// TIA Portal V17 export
// export: Created 2026-04-13T11:12:43.5207682Z, ExportSetting WithDefaults, DisplayName Totally Integrated Automation Portal, DisplayVersion V17 Update 4, DisplayName TIA Portal Openness, DisplayVersion V17 Update 4, DisplayName TIA Portal Version Control Interface, DisplayVersion V17, DisplayName SINAMICS Startdrive Advanced, DisplayVersion V17, DisplayName SINAMICS Startdrive G130, G150, S120, S150, SINAMICS MV, S210, DisplayVersion V17, DisplayName SINAMICS Startdrive G110M, G120, G120C, G120D, G120P, G115D, DisplayVersion V17, DisplayName STEP 7 Professional, DisplayVersion V17 Update 4, DisplayName STEP 7 Safety, DisplayVersion V17, DisplayName WinCC Professional, DisplayVersion V17 Update 4
FUNCTION_BLOCK "12放空阀"   // FB8, SCL
{ S7_Optimized_Access := 'FALSE' }
VERSION : 0.1
// stored: AutoNumber true, IsIECCheckEnabled false, SetENOAutomatically false, UDAEnableTagReadback false
   VAR_INPUT
      条件1 : Real;
      工程上限 : Real;
      工程下限 : Real;
      模拟高限 : Int;
      模拟低限 : Int;
   END_VAR
   VAR_IN_OUT
      模式设定 : Real;
      阀门启动 : Bool;
      阀门输出 : Bool;
      百分比设定值 : Real;
      输出百分比 : Int;
      PID反馈模拟量 : Int;
      YS映射到阀开度 : Real;
   END_VAR
   VAR DB_SPECIFIC
      动画 : Int;
      ST1 : Real;
   END_VAR
   VAR_TEMP
      TEMP_1 : Int;
   END_VAR
BEGIN
   // "IEC_Timer_0_DB".TON(IN:=#输出电源开,
   //                      PT:=T#10s,
   //                      Q=>  #阀开报警检测位);
   // IF #阀开报警检测位 AND #阀开信号  THEN
   //     #阀开异常报警 := TRUE;
   // ELSE
   //     #阀开异常报警 := FALSE;
   // END_IF;
   // "IEC_Timer_0_DB_1".TON (IN:=NOT #输出电源开,
   //                        PT:=T#10s,
   //                        Q=>#阀关报警检测位);
   // IF #阀关报警检测位 AND #阀关信号  THEN
   //     #阀关异常报警 := TRUE; ELSE
   //     #阀关异常报警 :=FALSE;
   // END_IF;
   //手动控制--------------------------------------------------------------------------------------------------------------
   IF #模式设定 = 2.0 THEN

       IF #阀门启动 THEN
           #阀门输出 := TRUE;
           #输出百分比 := REAL_TO_INT((#百分比设定值 - #工程下限) * (#模拟高限 - #模拟低限) / (#工程上限 - #工程下限) + #模拟低限);

       END_IF;
       IF NOT #阀门启动 THEN
           #阀门输出 := FALSE;
           #输出百分比 := REAL_TO_INT(#工程下限);

       END_IF;

   END_IF;

   // 自动启动--------------------------------------------------------------------------------------------------------------
   IF #阀门输出 AND #模式设定 = 1.0 THEN
       (* #输出百分比 := REAL_TO_INT((#百分比设定值 - #工程下限) * (#模拟高限 - #模拟低限) / (#工程上限 - #工程下限) + #模拟低限); *)


       #ST1 := NORM_X_REAL(MIN := 5530, VALUE := #输出百分比, MAX := 27648);
       #YS映射到阀开度 := SCALE_X_REAL(MIN := 0, VALUE := #ST1, MAX := 100);


   END_IF;
   IF NOT #阀门输出 THEN
       #YS映射到阀开度 := 0;
   END_IF;




   (* #TON1(IN := #电机输出 AND #电机电流 < 10,
                          PT := T#60s,
                          Q => #P1);

   IF #P1 OR #电机报警信号 THEN
       #电机报警输出 := TRUE;
   ELSE
       #电机报警输出 := FALSE;
   END_IF; *)



   IF #阀门输出  THEN
       IF "Clock_1Hz" THEN
           #TEMP_1 := #TEMP_1 + 1;
       END_IF;

       IF #TEMP_1 >= 3 THEN
           #TEMP_1 := 0;
       END_IF;
       IF #TEMP_1 < 1 THEN
           #动画 := 0;
       ELSE
           #动画 := 1;
       END_IF;

   END_IF;
   IF NOT #阀门输出 THEN
       #动画 := 0;
   END_IF;




   // IF #阀开异常报警 THEN
   //     #输出电源开 := FALSE;
   // END_IF;
   // IF #阀关异常报警 THEN
   //     #输出电源开 := TRUE;
   // END_IF;
END_FUNCTION_BLOCK
